// TIA Portal V19 export
TYPE "LAF_typeUnitStatus"
// Status of the unit
// stored: Access Published
   STRUCT
      acknowledgeActive : Bool;   // Acknowledge command active
      alarmsDisabled : Bool;   // Alarms disabled
      simulationActive : Bool;   // Simulation active
      safetyReleased : Bool;   // Safety released
      specialFunctions : "LAF_typeSpecialFunctions";   // Activated special functions
      mode : "LUC_typeModes";   // Current mode of the unit
      state : "LUC_typeStates";   // Current state of the unit
   END_STRUCT;
END_TYPE
